FUNCTION_BLOCK StartPauseResetButtons_HMI
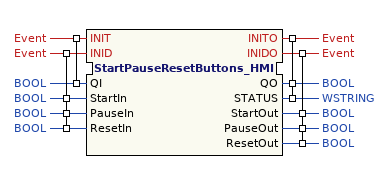
  EVENT_INPUT
    INIT WITH QI;
    INID WITH StartIn, PauseIn, ResetIn;
  END_EVENT
  EVENT_OUTPUT
    INITO WITH QO, STATUS;
    INIDO WITH StartOut, PauseOut, ResetOut;
  END_EVENT
  VAR_INPUT
    QI : BOOL;
    StartIn : BOOL;
    PauseIn : BOOL;
    ResetIn : BOOL;
  END_VAR
  VAR_OUTPUT
    QO : BOOL;
    STATUS : WSTRING;
    StartOut : BOOL;
    PauseOut : BOOL;
    ResetOut : BOOL;
  END_VAR
END_FUNCTION_BLOCK
